(* PLC project Tc2_Utilities.F_SwapRealEx Demo, tc3-libraries-kb TwinCAT 3.1 *)
(* stored: creationDateTime 2026-05-12T10:00:00, modificationDateTime 2026-05-12T10:00:00 *)

PROGRAM P_Demo_F_SwapRealEx
  VAR
    rTemperatureFromBc9000 : REAL := 1.5;  (* 通过 ADS 从 BC9000 读到的温度（带 BC 字节序） *)
    bSwapSucceeded : BOOL;  (* 交换成功标志（PDF 罕见返回 FALSE） *)
    bSwapRequest : BOOL;  (* 在线置 TRUE 触发一次字节序交换 *)
  END_VAR

// =============================================================================
// 场景：老工程改造——CX 控制器通过 ADS 从产线 BC9000 总线终端控制器读取
//       温度（REAL）数据上传 SCADA。BC9000 内存以"Hi-word 在前"存 REAL，
//       CX (x86/x64/Arm) 以"Lo-word 在前"存，直接读会得到完全错误的浮点值。
// 价值：手写 MEMCPY + WORD 交换 5 行容易在指针类型转换写错；本函数一次
//       调用、Beckhoff 验证、和 LREAL 版 F_SwapLRealEx 成套。
// 验证步骤：
//   1. 登录后 rTemperatureFromBc9000 = 1.5（4 字节内存 00 00 C0 3F，小端展示）。
//   2. 在线写 bSwapRequest := TRUE 触发交换。
//   3. 观察 rTemperatureFromBc9000 变为另一个值（约 -1.8e+38，因为按 BC
//      字节序解读 1.5 的内存是无意义浮点）；bSwapSucceeded = TRUE。
//   4. 重要：本函数是 INVOLUTION（双重交换=不交换）。再次触发，rTemperature
//      ...回到 1.5——印证 §3 的"两端各调一次会回到原值"。
//   5. 实际工程中：从 BC 读数据后只调一次，得到 PC 端正确值；写数据回 BC
//      前调一次，让 BC 收到的字节序对。
//   6. 注：新工程用 EtherCAT + IPC 不需要本函数，本例仅维护老项目时用。
// =============================================================================

IF bSwapRequest THEN
    // 单次调用：fVal 是 VAR_IN_OUT，原地修改
    bSwapSucceeded := F_SwapRealEx(fVal := rTemperatureFromBc9000);
    bSwapRequest := FALSE;
END_IF;
END_PROGRAM
